PROGRAM QUERYPOINTER
//__QUERYPOINTER
VAR
    iDerived   : I_Derived;
    fbVariante : FB_Variante;
    bResult    : BOOL;
    bTest      : BOOL;
    pFB        : POINTER TO FB_Variante;
END_VAR

//__QUERYPOINTER
iDerived := fbVariante;
bResult  := __QUERYPOINTER(iDerived, pFB);

IF bResult THEN
    bTest := pFB^.Derived();
END_IF

END_PROGRAM

(* stored: Version 1.1.0.1, ProductVersion 3.1.4024.12
   POU QUERYPOINTER: Id {9720a80e-d1de-4d43-aefa-ee7d76542c53}, SpecialFunc None *)
